{attribute addProperty BoxType "EL3773-0000-0019"}
{attribute addProperty Id "I1_SamplesAT %I*ARRAY [0..9] OF INT16020"}
{attribute addProperty CRC "2093022593"}
{attribute addProperty SizeInBites "160"}
{attribute addProperty SizeInBytes "20"}
TYPE L1_Current_Samples_7CC0FD81 :
STRUCT
	{attribute addProperty Name "I1_Samples"}
	I1_Samples AT %I* : ARRAY [0..9] OF INT;
END_STRUCT
END_TYPE

(* stored: Version 1.2.0.0, ProductVersion 3.1.4024.9
   DUT L1_Current_Samples_7CC0FD81: Id {b1fc7d4d-4a0c-4262-9bca-2872d65a7ec8} *)
